{attribute 'pack_mode' := '1'}
TYPE ST_DS402_6041h_StatusWord :
STRUCT
	b0_ReadyToSwitchOn 				: BIT; 
	b1_SwitchedOn 					: BIT; 
	b2_OperationEnabled 			: BIT; 
	b3_Fault						: BIT; 
	b4_VoltageEnabled				: BIT; 
	b5_QuickStop					: BIT;
	b6_SwitchOnDisabled				: BIT; 
	b7_Warning						: BIT; 
	b8_Synchranisation				: BIT; 
	b9_Remote						: BIT;
	b10_TargetReached				: BIT;
	b11_InternalLimitActive			: BIT; 
	b12_OperationModeSpecific		: BIT; 
	b13_OperationModeSpecific		: BIT; 
	b14_OperationModeSpecific		: BIT; 
	b15_ClosedLoopActive			: BIT;	
END_STRUCT
END_TYPE

(* stored: Version 1.1.0.1, ProductVersion 3.1.4024.12
   DUT ST_DS402_6041h_StatusWord: Id {c4cef78c-0a6c-0d9d-3bd5-153e0d96e255} *)
